FUNCTION_BLOCK POUc
VAR_INPUT
END_VAR
VAR_OUTPUT
END_VAR
VAR
END_VAR

END_FUNCTION_BLOCK

(* stored: Version 1.1.0.1, ProductVersion 3.1.0.26
   POU POUc: Id {d101945a-c89d-4f8c-bcc5-c3944e8509bf} *)
